FUNCTION_BLOCK FB_Foo
VAR_INPUT
	x : INT;
END_VAR


IF x < 5 THEN
	x := x + 1;
END_IF


METHOD PRIVATE m : DINT
VAR_INPUT
	r : REFERENCE TO INT;
END_VAR

VAR
	n : DINT;
END_VAR

n := 0;
// Count
WHILE r^ > 0 DO
	n := n + 1;
	r^ := r^ - 1;
END_WHILE

m := n;
END_METHOD

END_FUNCTION_BLOCK

(* stored: Version 1.1.0.1
   POU FB_Foo: Id {b}
   Method m: Id {c} *)
